INTERFACE I_Node EXTENDS I_Disposable, I_HostContent, I_HostInputPorts, I_HostOutputPorts, I_HostAlarms, I_HostParameters, I_HostExtensions, I_HostMetadata, I_EventEmitter, I_Deserializable, I_Serializable

METHOD PUBLIC Accept
VAR_INPUT
	Visitor : I_NodeVisitor;
END_VAR
END_METHOD

METHOD Clone : I_Node
VAR_INPUT
END_VAR
END_METHOD

METHOD PUBLIC Execute
END_METHOD

PROPERTY PUBLIC Id : T_MAXSTRING
GET
END_GET
END_PROPERTY

PROPERTY PUBLIC Mode : DINT
GET
END_GET
END_PROPERTY

PROPERTY PUBLIC Order : DINT
GET
END_GET
END_PROPERTY

END_INTERFACE

(* stored: Version 1.1.0.1, ProductVersion 3.1.4024.12
   Itf I_Node: Id {c7fe7db8-e5b5-493f-89de-ce411fbe90f1}
   Method Accept: Id {3b748c0f-1097-4f58-b766-99b78e1902fb}
   Method Clone: Id {5465cef7-3e38-4221-a083-2796d252cc4d}
   Method Execute: Id {ef78bbdf-aab1-403f-9e89-67287a1d445c}
   Property Id: Id {eca3800d-5167-4caf-95a2-3dc6470823d9}
   Get Get: Id {914f137a-939e-4208-8553-46cf7eafb463}
   Property Mode: Id {f796cc9f-66b6-4884-803a-b8002e8cab4f}
   Get Get: Id {bb35de38-10df-42a4-8101-66fce5da92c7}
   Property Order: Id {8a675645-2f7d-4226-aba0-aa7852e6360c}
   Get Get: Id {62f06775-93f4-46b5-807f-a64eeacc2f1d} *)
